// ---- DUTs/IO/Boxes/KL_C7B8B3CA.TcDUT
{attribute 'GeneratedUsingTerminal: KL3351-0003'}
{attribute addProperty BoxType "KL3351-0003"}
{attribute addProperty Description ""}
{attribute addProperty Physics ""}
{attribute addProperty Id "Channel_1AT %Q*Channel_0514A8FA0"}
{attribute addProperty CRC "3350770634"}
{attribute addProperty Size "0"}
TYPE KL_C7B8B3CA :
STRUCT
	{attribute addProperty Name "Channel_1"}
	Channel_1 : Channel_0514A8FA;
END_STRUCT
END_TYPE

// ---- DUTs/IO/Boxes/KL3356_E004D4E2.TcDUT
{attribute 'GeneratedUsingTerminal: KL3356'}
{attribute addProperty BoxType "KL3356"}
{attribute addProperty Description ""}
{attribute addProperty Physics ""}
{attribute addProperty Id "Channel_1AT %Q*Channel_4E9D1E2D0"}
{attribute addProperty CRC "3758413026"}
{attribute addProperty Size "0"}
TYPE KL3356_E004D4E2 :
STRUCT
	{attribute addProperty Name "Channel_1"}
	Channel_1 : Channel_4E9D1E2D;
END_STRUCT
END_TYPE

// ---- DUTs/IO/Boxes/KL_EE1D4506.TcDUT
{attribute 'GeneratedUsingTerminal: KL3361-0001'}
{attribute addProperty BoxType "KL3361-0001"}
{attribute addProperty Description ""}
{attribute addProperty Physics ""}
{attribute addProperty Id "Channel_1AT %Q*Channel_3C1A65000"}
{attribute addProperty CRC "3994895622"}
{attribute addProperty Size "0"}
TYPE KL_EE1D4506 :
STRUCT
	{attribute addProperty Name "Channel_1"}
	Channel_1 : Channel_3C1A6500;
END_STRUCT
END_TYPE

// ---- DUTs/IO/Boxes/KL3361_73CB82BA.TcDUT
{attribute 'GeneratedUsingTerminal: KL3361'}
{attribute addProperty BoxType "KL3361"}
{attribute addProperty Description ""}
{attribute addProperty Physics ""}
{attribute addProperty Id "Channel_1AT %Q*Channel_78571FB40"}
{attribute addProperty CRC "1942717114"}
{attribute addProperty Size "0"}
TYPE KL3361_73CB82BA :
STRUCT
	{attribute addProperty Name "Channel_1"}
	Channel_1 : Channel_78571FB4;
END_STRUCT
END_TYPE

// ---- DUTs/IO/Boxes/KL_73CB82BA.TcDUT
{attribute 'GeneratedUsingTerminal: KL3361-0003'}
{attribute addProperty BoxType "KL3361-0003"}
{attribute addProperty Description ""}
{attribute addProperty Physics ""}
{attribute addProperty Id "Channel_1AT %Q*Channel_78571FB40"}
{attribute addProperty CRC "1942717114"}
{attribute addProperty Size "0"}
TYPE KL_73CB82BA :
STRUCT
	{attribute addProperty Name "Channel_1"}
	Channel_1 : Channel_78571FB4;
END_STRUCT
END_TYPE

// ---- DUTs/IO/Boxes/KL3362_E98BF8F1.TcDUT
{attribute 'GeneratedUsingTerminal: KL3362'}
{attribute addProperty BoxType "KL3362"}
{attribute addProperty Description ""}
{attribute addProperty Physics ""}
{attribute addProperty Id "Channel_1AT %Q*Channel_3C1A65000Channel_2AT %Q*Channel_3C1A65000"}
{attribute addProperty CRC "3918264561"}
{attribute addProperty Size "0"}
TYPE KL3362_E98BF8F1 :
STRUCT
	{attribute addProperty Name "Channel_1"}
	Channel_1 : Channel_3C1A6500;
	{attribute addProperty Name "Channel_2"}
	Channel_2 : Channel_3C1A6500;
END_STRUCT
END_TYPE

// ---- DUTs/IO/Boxes/KL6211_60136EA1.TcDUT
{attribute 'GeneratedUsingTerminal: KL6211'}
{attribute addProperty BoxType "KL6211"}
{attribute addProperty Description ""}
{attribute addProperty Physics ""}
{attribute addProperty Id "Channel_1AT %Q*Channel_879058310"}
{attribute addProperty CRC "1611886241"}
{attribute addProperty Size "0"}
TYPE KL6211_60136EA1 :
STRUCT
	{attribute addProperty Name "Channel_1"}
	Channel_1 : Channel_87905831;
END_STRUCT
END_TYPE

// ---- DUTs/IO/Boxes/KL_9AE543B6.TcDUT
{attribute 'GeneratedUsingTerminal: KL6211-0020'}
{attribute addProperty BoxType "KL6211-0020"}
{attribute addProperty Description ""}
{attribute addProperty Physics ""}
{attribute addProperty Id "Channel_1AT %Q*Channel_099BCCDA0"}
{attribute addProperty CRC "2598716342"}
{attribute addProperty Size "0"}
TYPE KL_9AE543B6 :
STRUCT
	{attribute addProperty Name "Channel_1"}
	Channel_1 : Channel_099BCCDA;
END_STRUCT
END_TYPE

// ---- DUTs/IO/Boxes/KL_FC0201B8.TcDUT
{attribute 'GeneratedUsingTerminal: KL6211-0002'}
{attribute addProperty BoxType "KL6211-0002"}
{attribute addProperty Description ""}
{attribute addProperty Physics ""}
{attribute addProperty Id "Channel_1AT %Q*Channel_82ADD0760"}
{attribute addProperty CRC "4227989944"}
{attribute addProperty Size "0"}
TYPE KL_FC0201B8 :
STRUCT
	{attribute addProperty Name "Channel_1"}
	Channel_1 : Channel_82ADD076;
END_STRUCT
END_TYPE

// ---- DUTs/IO/Boxes/KL_498D8863.TcDUT
{attribute 'GeneratedUsingTerminal: KL6211-0022'}
{attribute addProperty BoxType "KL6211-0022"}
{attribute addProperty Description ""}
{attribute addProperty Physics ""}
{attribute addProperty Id "Channel_1AT %Q*Channel_332F026B0"}
{attribute addProperty CRC "1234012259"}
{attribute addProperty Size "0"}
TYPE KL_498D8863 :
STRUCT
	{attribute addProperty Name "Channel_1"}
	Channel_1 : Channel_332F026B;
END_STRUCT
END_TYPE

// ---- DUTs/IO/Boxes/KL_71341691.TcDUT
{attribute 'GeneratedUsingTerminal: KL6211-0004'}
{attribute addProperty BoxType "KL6211-0004"}
{attribute addProperty Description ""}
{attribute addProperty Physics ""}
{attribute addProperty Id "Channel_1AT %Q*Channel_A6A8AB450"}
{attribute addProperty CRC "1899239057"}
{attribute addProperty Size "0"}
TYPE KL_71341691 :
STRUCT
	{attribute addProperty Name "Channel_1"}
	Channel_1 : Channel_A6A8AB45;
END_STRUCT
END_TYPE

// ---- DUTs/IO/Boxes/KL_2B11657C.TcDUT
{attribute 'GeneratedUsingTerminal: KL6211-0024'}
{attribute addProperty BoxType "KL6211-0024"}
{attribute addProperty Description ""}
{attribute addProperty Physics ""}
{attribute addProperty Id "Channel_1AT %Q*Channel_A42BCA5C0"}
{attribute addProperty CRC "722560380"}
{attribute addProperty Size "0"}
TYPE KL_2B11657C :
STRUCT
	{attribute addProperty Name "Channel_1"}
	Channel_1 : Channel_A42BCA5C;
END_STRUCT
END_TYPE

// ---- DUTs/IO/Boxes/KL6224_C0F107BD.TcDUT
{attribute 'GeneratedUsingTerminal: KL6224'}
{attribute addProperty BoxType "KL6224"}
{attribute addProperty Description ""}
{attribute addProperty Physics ""}
{attribute addProperty Id "Channel_1AT %Q*Channel_08506BCE0"}
{attribute addProperty CRC "3237021629"}
{attribute addProperty Size "0"}
TYPE KL6224_C0F107BD :
STRUCT
	{attribute addProperty Name "Channel_1"}
	Channel_1 : Channel_08506BCE;
END_STRUCT
END_TYPE

// ---- DUTs/IO/Boxes/KL_FC1E3393.TcDUT
{attribute 'GeneratedUsingTerminal: KL6224-0001'}
{attribute addProperty BoxType "KL6224-0001"}
{attribute addProperty Description ""}
{attribute addProperty Physics ""}
{attribute addProperty Id "Channel_1AT %Q*Channel_085338040"}
{attribute addProperty CRC "4229837715"}
{attribute addProperty Size "0"}
TYPE KL_FC1E3393 :
STRUCT
	{attribute addProperty Name "Channel_1"}
	Channel_1 : Channel_08533804;
END_STRUCT
END_TYPE

// ---- DUTs/IO/Boxes/KL_C51B1CB0.TcDUT
{attribute 'GeneratedUsingTerminal: KL6224-0002'}
{attribute addProperty BoxType "KL6224-0002"}
{attribute addProperty Description ""}
{attribute addProperty Physics ""}
{attribute addProperty Id "Channel_1AT %Q*Channel_A04AC4BD0"}
{attribute addProperty CRC "3306888368"}
{attribute addProperty Size "0"}
TYPE KL_C51B1CB0 :
STRUCT
	{attribute addProperty Name "Channel_1"}
	Channel_1 : Channel_A04AC4BD;
END_STRUCT
END_TYPE

// ---- DUTs/IO/Boxes/KL_7EC2CD64.TcDUT
{attribute 'GeneratedUsingTerminal: KL6224-0003'}
{attribute addProperty BoxType "KL6224-0003"}
{attribute addProperty Description ""}
{attribute addProperty Physics ""}
{attribute addProperty Id "Channel_1AT %Q*Channel_779103830"}
{attribute addProperty CRC "2126695780"}
{attribute addProperty Size "0"}
TYPE KL_7EC2CD64 :
STRUCT
	{attribute addProperty Name "Channel_1"}
	Channel_1 : Channel_77910383;
END_STRUCT
END_TYPE

// ---- DUTs/IO/Boxes/KL_3829421A.TcDUT
{attribute 'GeneratedUsingTerminal: KL6301-0002'}
{attribute addProperty BoxType "KL6301-0002"}
{attribute addProperty Description ""}
{attribute addProperty Physics ""}
{attribute addProperty Id "Channel_1AT %Q*Channel_9BC0092E0"}
{attribute addProperty CRC "942227994"}
{attribute addProperty Size "0"}
TYPE KL_3829421A :
STRUCT
	{attribute addProperty Name "Channel_1"}
	Channel_1 : Channel_9BC0092E;
END_STRUCT
END_TYPE

// ---- DUTs/IO/Boxes/KL_9116C2C1.TcDUT
{attribute 'GeneratedUsingTerminal: KL6401-0002'}
{attribute addProperty BoxType "KL6401-0002"}
{attribute addProperty Description ""}
{attribute addProperty Physics ""}
{attribute addProperty Id "Channel_1AT %Q*Channel_7606D9890"}
{attribute addProperty CRC "2434187969"}
{attribute addProperty Size "0"}
TYPE KL_9116C2C1 :
STRUCT
	{attribute addProperty Name "Channel_1"}
	Channel_1 : Channel_7606D989;
END_STRUCT
END_TYPE

// ---- DUTs/IO/Boxes/KL6551_528AE398.TcDUT
{attribute 'GeneratedUsingTerminal: KL6551'}
{attribute addProperty BoxType "KL6551"}
{attribute addProperty Description ""}
{attribute addProperty Physics ""}
{attribute addProperty Id "Channel_1AT %Q*Channel_6931CC5B0"}
{attribute addProperty CRC "1384833944"}
{attribute addProperty Size "0"}
TYPE KL6551_528AE398 :
STRUCT
	{attribute addProperty Name "Channel_1"}
	Channel_1 : Channel_6931CC5B;
END_STRUCT
END_TYPE

// ---- DUTs/IO/Boxes/KL_3325E583.TcDUT
{attribute 'GeneratedUsingTerminal: KL6581-0002'}
{attribute addProperty BoxType "KL6581-0002"}
{attribute addProperty Description ""}
{attribute addProperty Physics ""}
{attribute addProperty Id "Channel_1AT %Q*Channel_F7FDEFA00"}
{attribute addProperty CRC "858121603"}
{attribute addProperty Size "0"}
TYPE KL_3325E583 :
STRUCT
	{attribute addProperty Name "Channel_1"}
	Channel_1 : Channel_F7FDEFA0;
END_STRUCT
END_TYPE

// ---- DUTs/IO/Boxes/KL_528AE398.TcDUT
{attribute 'GeneratedUsingTerminal: KL6771-0002'}
{attribute addProperty BoxType "KL6771-0002"}
{attribute addProperty Description ""}
{attribute addProperty Physics ""}
{attribute addProperty Id "Channel_1AT %Q*Channel_6931CC5B0"}
{attribute addProperty CRC "1384833944"}
{attribute addProperty Size "0"}
TYPE KL_528AE398 :
STRUCT
	{attribute addProperty Name "Channel_1"}
	Channel_1 : Channel_6931CC5B;
END_STRUCT
END_TYPE

// ---- DUTs/IO/Boxes/KL6781_BE595CA2.TcDUT
{attribute 'GeneratedUsingTerminal: KL6781'}
{attribute addProperty BoxType "KL6781"}
{attribute addProperty Description ""}
{attribute addProperty Physics ""}
{attribute addProperty Id "Channel_1AT %Q*Channel_A1C14FB40"}
{attribute addProperty CRC "3193527458"}
{attribute addProperty Size "0"}
TYPE KL6781_BE595CA2 :
STRUCT
	{attribute addProperty Name "Channel_1"}
	Channel_1 : Channel_A1C14FB4;
END_STRUCT
END_TYPE

// ---- DUTs/IO/Boxes/KL6811_6148C904.TcDUT
{attribute 'GeneratedUsingTerminal: KL6811'}
{attribute addProperty BoxType "KL6811"}
{attribute addProperty Description ""}
{attribute addProperty Physics ""}
{attribute addProperty Id "Channel_1AT %Q*Channel_6576A6810"}
{attribute addProperty CRC "1632160004"}
{attribute addProperty Size "0"}
TYPE KL6811_6148C904 :
STRUCT
	{attribute addProperty Name "Channel_1"}
	Channel_1 : Channel_6576A681;
END_STRUCT
END_TYPE

// ---- DUTs/IO/Boxes/KL6821_F77C82D2.TcDUT
{attribute 'GeneratedUsingTerminal: KL6821'}
{attribute addProperty BoxType "KL6821"}
{attribute addProperty Description ""}
{attribute addProperty Physics ""}
{attribute addProperty Id "Channel_1AT %Q*Channel_A4B48F2D0"}
{attribute addProperty CRC "4152132306"}
{attribute addProperty Size "0"}
TYPE KL6821_F77C82D2 :
STRUCT
	{attribute addProperty Name "Channel_1"}
	Channel_1 : Channel_A4B48F2D;
END_STRUCT
END_TYPE

// ---- DUTs/IO/Boxes/KL6831_BE595CA2.TcDUT
{attribute 'GeneratedUsingTerminal: KL6831'}
{attribute addProperty BoxType "KL6831"}
{attribute addProperty Description ""}
{attribute addProperty Physics ""}
{attribute addProperty Id "Channel_1AT %Q*Channel_A1C14FB40"}
{attribute addProperty CRC "3193527458"}
{attribute addProperty Size "0"}
TYPE KL6831_BE595CA2 :
STRUCT
	{attribute addProperty Name "Channel_1"}
	Channel_1 : Channel_A1C14FB4;
END_STRUCT
END_TYPE

// ---- DUTs/IO/Boxes/KL6841_BE595CA2.TcDUT
{attribute 'GeneratedUsingTerminal: KL6841'}
{attribute addProperty BoxType "KL6841"}
{attribute addProperty Description ""}
{attribute addProperty Physics ""}
{attribute addProperty Id "Channel_1AT %Q*Channel_A1C14FB40"}
{attribute addProperty CRC "3193527458"}
{attribute addProperty Size "0"}
TYPE KL6841_BE595CA2 :
STRUCT
	{attribute addProperty Name "Channel_1"}
	Channel_1 : Channel_A1C14FB4;
END_STRUCT
END_TYPE

// ---- DUTs/IO/Boxes/KL6904_B938D612.TcDUT
{attribute 'GeneratedUsingTerminal: KL6904'}
{attribute addProperty BoxType "KL6904"}
{attribute addProperty Description ""}
{attribute addProperty Physics ""}
{attribute addProperty Id "Channel_1AT %Q*Channel_9E2936860"}
{attribute addProperty CRC "3107509778"}
{attribute addProperty Size "0"}
TYPE KL6904_B938D612 :
STRUCT
	{attribute addProperty Name "Channel_1"}
	Channel_1 : Channel_9E293686;
END_STRUCT
END_TYPE

// ---- DUTs/IO/Boxes/KL_921B772D.TcDUT
{attribute 'GeneratedUsingTerminal: KL6904-0001'}
{attribute addProperty BoxType "KL6904-0001"}
{attribute addProperty Description ""}
{attribute addProperty Physics ""}
{attribute addProperty Id "Channel_1AT %Q*Channel_F84AC14F0"}
{attribute addProperty CRC "2451273517"}
{attribute addProperty Size "0"}
TYPE KL_921B772D :
STRUCT
	{attribute addProperty Name "Channel_1"}
	Channel_1 : Channel_F84AC14F;
END_STRUCT
END_TYPE

// ---- DUTs/IO/Boxes/KL_779990DF.TcDUT
{attribute 'GeneratedUsingTerminal: KL8001-0002'}
{attribute addProperty BoxType "KL8001-0002"}
{attribute addProperty Description ""}
{attribute addProperty Physics ""}
{attribute addProperty Id "Channel_1AT %Q*Channel_2F3145090"}
{attribute addProperty CRC "2006552799"}
{attribute addProperty Size "0"}
TYPE KL_779990DF :
STRUCT
	{attribute addProperty Name "Channel_1"}
	Channel_1 : Channel_2F314509;
END_STRUCT
END_TYPE

// ---- DUTs/IO/Boxes/KL8001_7761653A.TcDUT
{attribute 'GeneratedUsingTerminal: KL8001'}
{attribute addProperty BoxType "KL8001"}
{attribute addProperty Description ""}
{attribute addProperty Physics ""}
{attribute addProperty Id "Channel_1AT %Q*Channel_D9D488070"}
{attribute addProperty CRC "2002871610"}
{attribute addProperty Size "0"}
TYPE KL8001_7761653A :
STRUCT
	{attribute addProperty Name "Channel_1"}
	Channel_1 : Channel_D9D48807;
END_STRUCT
END_TYPE

// ---- DUTs/IO/Boxes/KL8519_8C34650F.TcDUT
{attribute 'GeneratedUsingTerminal: KL8519'}
{attribute addProperty BoxType "KL8519"}
{attribute addProperty Description ""}
{attribute addProperty Physics ""}
{attribute addProperty Id "Channel_1AT %Q*Channel_D13646E30"}
{attribute addProperty CRC "2352243983"}
{attribute addProperty Size "0"}
TYPE KL8519_8C34650F :
STRUCT
	{attribute addProperty Name "Channel_1"}
	Channel_1 : Channel_D13646E3;
END_STRUCT
END_TYPE

// ---- DUTs/IO/Boxes/KL8524_A4B9216E.TcDUT
{attribute 'GeneratedUsingTerminal: KL8524'}
{attribute addProperty BoxType "KL8524"}
{attribute addProperty Description ""}
{attribute addProperty Physics ""}
{attribute addProperty Id "Channel_1AT %Q*Channel_3263D8D50"}
{attribute addProperty CRC "2763596142"}
{attribute addProperty Size "0"}
TYPE KL8524_A4B9216E :
STRUCT
	{attribute addProperty Name "Channel_1"}
	Channel_1 : Channel_3263D8D5;
END_STRUCT
END_TYPE

// ---- DUTs/IO/Boxes/KL8528_73A97EC1.TcDUT
{attribute 'GeneratedUsingTerminal: KL8528'}
{attribute addProperty BoxType "KL8528"}
{attribute addProperty Description ""}
{attribute addProperty Physics ""}
{attribute addProperty Id "Channel_1AT %Q*Channel_D490E9730"}
{attribute addProperty CRC "1940487873"}
{attribute addProperty Size "0"}
TYPE KL8528_73A97EC1 :
STRUCT
	{attribute addProperty Name "Channel_1"}
	Channel_1 : Channel_D490E973;
END_STRUCT
END_TYPE

// ---- DUTs/IO/Boxes/KL8548_23451728.TcDUT
{attribute 'GeneratedUsingTerminal: KL8548'}
{attribute addProperty BoxType "KL8548"}
{attribute addProperty Description ""}
{attribute addProperty Physics ""}
{attribute addProperty Id "Channel_1AT %Q*Channel_6576A6810Channel_2AT %Q*Channel_6576A6810Channel_3AT %Q*Channel_6576A6810Channel_4AT %Q*Channel_6576A6810Channel_5AT %Q*Channel_6576A6810Channel_6AT %Q*Channel_6576A6810Channel_7AT %Q*Channel_6576A6810Channel_8AT %Q*Channel_6576A6810"}
{attribute addProperty CRC "591730472"}
{attribute addProperty Size "0"}
TYPE KL8548_23451728 :
STRUCT
	{attribute addProperty Name "Channel_1"}
	Channel_1 : Channel_6576A681;
	{attribute addProperty Name "Channel_2"}
	Channel_2 : Channel_6576A681;
	{attribute addProperty Name "Channel_3"}
	Channel_3 : Channel_6576A681;
	{attribute addProperty Name "Channel_4"}
	Channel_4 : Channel_6576A681;
	{attribute addProperty Name "Channel_5"}
	Channel_5 : Channel_6576A681;
	{attribute addProperty Name "Channel_6"}
	Channel_6 : Channel_6576A681;
	{attribute addProperty Name "Channel_7"}
	Channel_7 : Channel_6576A681;
	{attribute addProperty Name "Channel_8"}
	Channel_8 : Channel_6576A681;
END_STRUCT
END_TYPE

// ---- DUTs/IO/Boxes/KL8610_C571D068.TcDUT
{attribute 'GeneratedUsingTerminal: KL8610'}
{attribute addProperty BoxType "KL8610"}
{attribute addProperty Description ""}
{attribute addProperty Physics ""}
{attribute addProperty Id "KL8601_1AT %Q*KL_6576A6810"}
{attribute addProperty CRC "3312570472"}
{attribute addProperty Size "0"}
TYPE KL8610_C571D068 :
STRUCT
	{attribute addProperty Name "KL8601_1"}
	KL8601_1 : KL_6576A681;
END_STRUCT
END_TYPE

// ---- DUTs/IO/Boxes/KL_5A83E84C.TcDUT
{attribute 'GeneratedUsingTerminal: KL8610-0001'}
{attribute addProperty BoxType "KL8610-0001"}
{attribute addProperty Description ""}
{attribute addProperty Physics ""}
{attribute addProperty Id "KL8601_1AT %Q*KL_6576A6810KL8601_2AT %Q*KL_6576A6810"}
{attribute addProperty CRC "1518594124"}
{attribute addProperty Size "0"}
TYPE KL_5A83E84C :
STRUCT
	{attribute addProperty Name "KL8601_1"}
	KL8601_1 : KL_6576A681;
	{attribute addProperty Name "KL8601_2"}
	KL8601_2 : KL_6576A681;
END_STRUCT
END_TYPE

// ---- DUTs/IO/Boxes/KL_BF4AA06C.TcDUT
{attribute 'GeneratedUsingTerminal: KL8610-0002'}
{attribute addProperty BoxType "KL8610-0002"}
{attribute addProperty Description ""}
{attribute addProperty Physics ""}
{attribute addProperty Id "KL8601_1AT %Q*KL_6576A6810KL8601_2AT %Q*KL_6576A6810KL8601_3AT %Q*KL_6576A6810"}
{attribute addProperty CRC "3209338988"}
{attribute addProperty Size "0"}
TYPE KL_BF4AA06C :
STRUCT
	{attribute addProperty Name "KL8601_1"}
	KL8601_1 : KL_6576A681;
	{attribute addProperty Name "KL8601_2"}
	KL8601_2 : KL_6576A681;
	{attribute addProperty Name "KL8601_3"}
	KL8601_3 : KL_6576A681;
END_STRUCT
END_TYPE

// ---- DUTs/IO/Boxes/KL_7485E925.TcDUT
{attribute 'GeneratedUsingTerminal: KL8610-0003'}
{attribute addProperty BoxType "KL8610-0003"}
{attribute addProperty Description ""}
{attribute addProperty Physics ""}
{attribute addProperty Id "KL8601_1AT %Q*KL_6576A6810KL8601_2AT %Q*KL_6576A6810KL8601_3AT %Q*KL_6576A6810KL8601_4AT %Q*KL_6576A6810"}
{attribute addProperty CRC "1954933029"}
{attribute addProperty Size "0"}
TYPE KL_7485E925 :
STRUCT
	{attribute addProperty Name "KL8601_1"}
	KL8601_1 : KL_6576A681;
	{attribute addProperty Name "KL8601_2"}
	KL8601_2 : KL_6576A681;
	{attribute addProperty Name "KL8601_3"}
	KL8601_3 : KL_6576A681;
	{attribute addProperty Name "KL8601_4"}
	KL8601_4 : KL_6576A681;
END_STRUCT
END_TYPE

// ---- DUTs/IO/Boxes/KL_372C6BEC.TcDUT
{attribute 'GeneratedUsingTerminal: KL8610-0004'}
{attribute addProperty BoxType "KL8610-0004"}
{attribute addProperty Description ""}
{attribute addProperty Physics ""}
{attribute addProperty Id "KL8601_1AT %Q*KL_6576A6810KL8601_2AT %Q*KL_6576A6810KL8601_3AT %Q*KL_6576A6810KL8601_4AT %Q*KL_6576A6810KL8601_5AT %Q*KL_6576A6810"}
{attribute addProperty CRC "925658092"}
{attribute addProperty Size "0"}
TYPE KL_372C6BEC :
STRUCT
	{attribute addProperty Name "KL8601_1"}
	KL8601_1 : KL_6576A681;
	{attribute addProperty Name "KL8601_2"}
	KL8601_2 : KL_6576A681;
	{attribute addProperty Name "KL8601_3"}
	KL8601_3 : KL_6576A681;
	{attribute addProperty Name "KL8601_4"}
	KL8601_4 : KL_6576A681;
	{attribute addProperty Name "KL8601_5"}
	KL8601_5 : KL_6576A681;
END_STRUCT
END_TYPE

// ---- DUTs/IO/Boxes/KL_2E5CD6C8.TcDUT
{attribute 'GeneratedUsingTerminal: KL8610-0005'}
{attribute addProperty BoxType "KL8610-0005"}
{attribute addProperty Description ""}
{attribute addProperty Physics ""}
{attribute addProperty Id "KL8601_1AT %Q*KL_6576A6810KL8601_2AT %Q*KL_6576A6810KL8601_3AT %Q*KL_6576A6810KL8601_4AT %Q*KL_6576A6810KL8601_5AT %Q*KL_6576A6810KL8601_6AT %Q*KL_6576A6810"}
{attribute addProperty CRC "777836232"}
{attribute addProperty Size "0"}
TYPE KL_2E5CD6C8 :
STRUCT
	{attribute addProperty Name "KL8601_1"}
	KL8601_1 : KL_6576A681;
	{attribute addProperty Name "KL8601_2"}
	KL8601_2 : KL_6576A681;
	{attribute addProperty Name "KL8601_3"}
	KL8601_3 : KL_6576A681;
	{attribute addProperty Name "KL8601_4"}
	KL8601_4 : KL_6576A681;
	{attribute addProperty Name "KL8601_5"}
	KL8601_5 : KL_6576A681;
	{attribute addProperty Name "KL8601_6"}
	KL8601_6 : KL_6576A681;
END_STRUCT
END_TYPE

// ---- DUTs/IO/Boxes/KL_68BDE1E9.TcDUT
{attribute 'GeneratedUsingTerminal: KL8610-0006'}
{attribute addProperty BoxType "KL8610-0006"}
{attribute addProperty Description ""}
{attribute addProperty Physics ""}
{attribute addProperty Id "KL8601_1AT %Q*KL_6576A6810KL8601_2AT %Q*KL_6576A6810KL8601_3AT %Q*KL_6576A6810KL8601_4AT %Q*KL_6576A6810KL8601_5AT %Q*KL_6576A6810KL8601_6AT %Q*KL_6576A6810KL8601_7AT %Q*KL_6576A6810"}
{attribute addProperty CRC "1757274601"}
{attribute addProperty Size "0"}
TYPE KL_68BDE1E9 :
STRUCT
	{attribute addProperty Name "KL8601_1"}
	KL8601_1 : KL_6576A681;
	{attribute addProperty Name "KL8601_2"}
	KL8601_2 : KL_6576A681;
	{attribute addProperty Name "KL8601_3"}
	KL8601_3 : KL_6576A681;
	{attribute addProperty Name "KL8601_4"}
	KL8601_4 : KL_6576A681;
	{attribute addProperty Name "KL8601_5"}
	KL8601_5 : KL_6576A681;
	{attribute addProperty Name "KL8601_6"}
	KL8601_6 : KL_6576A681;
	{attribute addProperty Name "KL8601_7"}
	KL8601_7 : KL_6576A681;
END_STRUCT
END_TYPE

// ---- DUTs/IO/Boxes/KL_84AAE8B6.TcDUT
{attribute 'GeneratedUsingTerminal: KL8610-0007'}
{attribute addProperty BoxType "KL8610-0007"}
{attribute addProperty Description ""}
{attribute addProperty Physics ""}
{attribute addProperty Id "KL8601_1AT %Q*KL_6576A6810KL8601_2AT %Q*KL_6576A6810KL8601_3AT %Q*KL_6576A6810KL8601_4AT %Q*KL_6576A6810KL8601_5AT %Q*KL_6576A6810KL8601_6AT %Q*KL_6576A6810KL8601_7AT %Q*KL_6576A6810KL8601_8AT %Q*KL_6576A6810"}
{attribute addProperty CRC "2225793206"}
{attribute addProperty Size "0"}
TYPE KL_84AAE8B6 :
STRUCT
	{attribute addProperty Name "KL8601_1"}
	KL8601_1 : KL_6576A681;
	{attribute addProperty Name "KL8601_2"}
	KL8601_2 : KL_6576A681;
	{attribute addProperty Name "KL8601_3"}
	KL8601_3 : KL_6576A681;
	{attribute addProperty Name "KL8601_4"}
	KL8601_4 : KL_6576A681;
	{attribute addProperty Name "KL8601_5"}
	KL8601_5 : KL_6576A681;
	{attribute addProperty Name "KL8601_6"}
	KL8601_6 : KL_6576A681;
	{attribute addProperty Name "KL8601_7"}
	KL8601_7 : KL_6576A681;
	{attribute addProperty Name "KL8601_8"}
	KL8601_8 : KL_6576A681;
END_STRUCT
END_TYPE

// ---- DUTs/IO/Boxes/KL9110_8BEE55F2.TcDUT
{attribute 'GeneratedUsingTerminal: KL9110'}
{attribute addProperty BoxType "KL9110"}
{attribute addProperty Description ""}
{attribute addProperty Physics ""}
{attribute addProperty Id "Channel_1AT %I*Channel_64AAC8C70"}
{attribute addProperty CRC "2347652594"}
{attribute addProperty Size "0"}
TYPE KL9110_8BEE55F2 :
STRUCT
	{attribute addProperty Name "Channel_1"}
	Channel_1 : Channel_64AAC8C7;
END_STRUCT
END_TYPE

// ---- DUTs/IO/Boxes/KL9160_8BEE55F2.TcDUT
{attribute 'GeneratedUsingTerminal: KL9160'}
{attribute addProperty BoxType "KL9160"}
{attribute addProperty Description ""}
{attribute addProperty Physics ""}
{attribute addProperty Id "Channel_1AT %I*Channel_64AAC8C70"}
{attribute addProperty CRC "2347652594"}
{attribute addProperty Size "0"}
TYPE KL9160_8BEE55F2 :
STRUCT
	{attribute addProperty Name "Channel_1"}
	Channel_1 : Channel_64AAC8C7;
END_STRUCT
END_TYPE

// ---- DUTs/IO/Boxes/KL9191_962A24DF.TcDUT
{attribute 'GeneratedUsingTerminal: KL9191'}
{attribute addProperty BoxType "KL9191"}
{attribute addProperty Description ""}
{attribute addProperty Physics ""}
{attribute addProperty Id "Channel_1AT %Q*Channel_471FAA5C0"}
{attribute addProperty CRC "2519344351"}
{attribute addProperty Size "0"}
TYPE KL9191_962A24DF :
STRUCT
	{attribute addProperty Name "Channel_1"}
	Channel_1 : Channel_471FAA5C;
END_STRUCT
END_TYPE

// ---- DUTs/IO/Boxes/KL9210_8BEE55F2.TcDUT
{attribute 'GeneratedUsingTerminal: KL9210'}
{attribute addProperty BoxType "KL9210"}
{attribute addProperty Description ""}
{attribute addProperty Physics ""}
{attribute addProperty Id "Channel_1AT %I*Channel_64AAC8C70"}
{attribute addProperty CRC "2347652594"}
{attribute addProperty Size "0"}
TYPE KL9210_8BEE55F2 :
STRUCT
	{attribute addProperty Name "Channel_1"}
	Channel_1 : Channel_64AAC8C7;
END_STRUCT
END_TYPE

// ---- DUTs/IO/Boxes/KL9260_8BEE55F2.TcDUT
{attribute 'GeneratedUsingTerminal: KL9260'}
{attribute addProperty BoxType "KL9260"}
{attribute addProperty Description ""}
{attribute addProperty Physics ""}
{attribute addProperty Id "Channel_1AT %I*Channel_64AAC8C70"}
{attribute addProperty CRC "2347652594"}
{attribute addProperty Size "0"}
TYPE KL9260_8BEE55F2 :
STRUCT
	{attribute addProperty Name "Channel_1"}
	Channel_1 : Channel_64AAC8C7;
END_STRUCT
END_TYPE

// ---- DUTs/IO/Boxes/KL_E4BD2B38.TcDUT
{attribute 'GeneratedUsingTerminal: KL9505-0010'}
{attribute addProperty BoxType "KL9505-0010"}
{attribute addProperty Description ""}
{attribute addProperty Physics ""}
{attribute addProperty Id "Diag_1AT %I*Diag_1F4F45730"}
{attribute addProperty CRC "3837602616"}
{attribute addProperty Size "0"}
TYPE KL_E4BD2B38 :
STRUCT
	{attribute addProperty Name "Diag_1"}
	Diag_1 : Diag_1F4F4573;
END_STRUCT
END_TYPE

// ---- DUTs/IO/Boxes/KL9528_8C984603.TcDUT
{attribute 'GeneratedUsingTerminal: KL9528'}
{attribute addProperty BoxType "KL9528"}
{attribute addProperty Description ""}
{attribute addProperty Physics ""}
{attribute addProperty Id "Channel_1AT %Q*Channel_0029832E0"}
{attribute addProperty CRC "2358789635"}
{attribute addProperty Size "0"}
TYPE KL9528_8C984603 :
STRUCT
	{attribute addProperty Name "Channel_1"}
	Channel_1 : Channel_0029832E;
END_STRUCT
END_TYPE

// ---- DUTs/IO/Boxes/KL9999_7A10A7F6.TcDUT
{attribute 'GeneratedUsingTerminal: KL9999'}
{attribute addProperty BoxType "KL9999"}
{attribute addProperty Description ""}
{attribute addProperty Physics ""}
{attribute addProperty Id "Channel_1AT %Q*Channel_126527430"}
{attribute addProperty CRC "2047911926"}
{attribute addProperty Size "0"}
TYPE KL9999_7A10A7F6 :
STRUCT
	{attribute addProperty Name "Channel_1"}
	Channel_1 : Channel_12652743;
END_STRUCT
END_TYPE

// ---- DUTs/IO/Devices/SyncUnitTask_2D604ED5.TcDUT
{attribute 'GeneratedUsingTerminal: IODEVICETYPE_ETHERCATPROT'}
{attribute addProperty BoxType "IODEVICETYPE_ETHERCATPROT"}
{attribute addProperty Id "WcStateAT %I*WcState_0B2B16F91InfoDataAT %I*InfoData_2A97D6CF8"}
{attribute addProperty CRC "761286357"}
{attribute addProperty Size "9"}
TYPE SyncUnitTask_2D604ED5 :
STRUCT
	{attribute addProperty Name "WcState"}
	WcState : WcState_0B2B16F9;
	{attribute addProperty Name "InfoData"}
	InfoData : InfoData_2A97D6CF;
END_STRUCT
END_TYPE

// ---- DUTs/IO/Devices/SyncUnitTasks_6FEB8257.TcDUT
{attribute 'GeneratedUsingTerminal: '}
{attribute addProperty BoxType ""}
{attribute addProperty Id "unreferencedAT %I*SyncUnitTask_2D604ED59PlcTaskAT %I*SyncUnitTask_2D604ED59"}
{attribute addProperty CRC "1877705303"}
{attribute addProperty Size "18"}
TYPE SyncUnitTasks_6FEB8257 :
STRUCT
	{attribute addProperty Name "unreferenced"}
	unreferenced : SyncUnitTask_2D604ED5;
	{attribute addProperty Name "PlcTask"}
	PlcTask : SyncUnitTask_2D604ED5;
END_STRUCT
END_TYPE

// ---- DUTs/IO/Devices/SyncUnits_99E584AF.TcDUT
{attribute 'GeneratedUsingTerminal: '}
{attribute addProperty BoxType ""}
{attribute addProperty Id "_defaultAT %I*SyncUnitTasks_6FEB825718"}
{attribute addProperty CRC "2581955759"}
{attribute addProperty Size "18"}
TYPE SyncUnits_99E584AF :
STRUCT
	{attribute addProperty Name "_default"}
	_default : SyncUnitTasks_6FEB8257;
END_STRUCT
END_TYPE

// ---- DUTs/IO/Topology/A_0014_BK1250_0000_0000_09E1EB45.TcDUT
{attribute 'GeneratedUsingTerminal: BK1250-0000-0000'}
{attribute addProperty BoxType "BK1250-0000-0000"}
{attribute addProperty Id "Term_397_KL1002KL1002_BB38DA8F0"}
{attribute addProperty CRC "165800773"}
{attribute addProperty Size "0"}
{attribute addProperty Name "A_0014(BK1250-0000-0000)"}
TYPE A_0014_BK1250_0000_0000_09E1EB45 EXTENDS BK1250_A2FCADE7 :
STRUCT
	{attribute addProperty Name "Term_397_KL1002"}
	Term_397_KL1002 : KL1002_BB38DA8F;
END_STRUCT
END_TYPE

// ---- DUTs/IO/Topology/Beckhoff_BKxxxxsub_EK1100_59A46924.TcDUT
{attribute 'GeneratedUsingTerminal: EK1100-0000-0018'}
{attribute addProperty BoxType "EK1100-0000-0018"}
{attribute addProperty Id "A_0014_BK1250_0000_0000A_0014_BK1250_0000_0000_09E1EB450"}
{attribute addProperty CRC "1503947044"}
{attribute addProperty Size "0"}
{attribute addProperty Name "Beckhoff BKxxxxsub EK1100"}
TYPE Beckhoff_BKxxxxsub_EK1100_59A46924 EXTENDS EK1100_1FC0878B :
STRUCT
	{attribute addProperty Name "A_0014(BK1250-0000-0000)"}
	{attribute addProperty PreviousPort "Beckhoff BKxxxxsub EK1100 : B"}
	A_0014_BK1250_0000_0000 : A_0014_BK1250_0000_0000_09E1EB45;
END_STRUCT
END_TYPE

// ---- DUTs/IO/Topology/A_0001_BK1120_0000_0000_205E6559.TcDUT
{attribute 'GeneratedUsingTerminal: BK1120-0000-0000'}
{attribute addProperty BoxType "BK1120-0000-0000"}
{attribute addProperty Id "Term_374_KL1002KL1002_BB38DA8F0"}
{attribute addProperty CRC "543057241"}
{attribute addProperty Size "0"}
{attribute addProperty Name "A_0001(BK1120-0000-0000)"}
TYPE A_0001_BK1120_0000_0000_205E6559 EXTENDS BK1120_6D44499E :
STRUCT
	{attribute addProperty Name "Term_374_KL1002"}
	Term_374_KL1002 : KL1002_BB38DA8F;
END_STRUCT
END_TYPE

// ---- DUTs/IO/Topology/A_0002_BK1120_0000_0001_76F1F8EB.TcDUT
{attribute 'GeneratedUsingTerminal: BK1120-0000-0001'}
{attribute addProperty BoxType "BK1120-0000-0001"}
{attribute addProperty Id "Term_375_KL1002KL1002_BB38DA8F0"}
{attribute addProperty CRC "1995569387"}
{attribute addProperty Size "0"}
{attribute addProperty Name "A_0002(BK1120-0000-0001)"}
TYPE A_0002_BK1120_0000_0001_76F1F8EB EXTENDS BK1120_A2FCADE7 :
STRUCT
	{attribute addProperty Name "Term_375_KL1002"}
	Term_375_KL1002 : KL1002_BB38DA8F;
END_STRUCT
END_TYPE

// ---- DUTs/IO/Topology/A_0003_BK1120_0000_0016_8D015E3D.TcDUT
{attribute 'GeneratedUsingTerminal: BK1120-0000-0016'}
{attribute addProperty BoxType "BK1120-0000-0016"}
{attribute addProperty Id "Term_376_KL1002KL1002_BB38DA8F0"}
{attribute addProperty CRC "2365677117"}
{attribute addProperty Size "0"}
{attribute addProperty Name "A_0003(BK1120-0000-0016)"}
TYPE A_0003_BK1120_0000_0016_8D015E3D EXTENDS BK1120_A2FCADE7 :
STRUCT
	{attribute addProperty Name "Term_376_KL1002"}
	Term_376_KL1002 : KL1002_BB38DA8F;
END_STRUCT
END_TYPE

// ---- DUTs/IO/Topology/A_0004_BK1120_0000_0017_DBAEC38F.TcDUT
{attribute 'GeneratedUsingTerminal: BK1120-0000-0017'}
{attribute addProperty BoxType "BK1120-0000-0017"}
{attribute addProperty Id "Term_377_KL1002KL1002_BB38DA8F0"}
{attribute addProperty CRC "3685663631"}
{attribute addProperty Size "0"}
{attribute addProperty Name "A_0004(BK1120-0000-0017)"}
TYPE A_0004_BK1120_0000_0017_DBAEC38F EXTENDS BK1120_A2FCADE7 :
STRUCT
	{attribute addProperty Name "Term_377_KL1002"}
	Term_377_KL1002 : KL1002_BB38DA8F;
END_STRUCT
END_TYPE

// ---- DUTs/IO/Topology/A_0005_BK1120_0000_0018_C2DFD8D8.TcDUT
{attribute 'GeneratedUsingTerminal: BK1120-0000-0018'}
{attribute addProperty BoxType "BK1120-0000-0018"}
{attribute addProperty Id "Term_378_KL1002KL1002_BB38DA8F0"}
{attribute addProperty CRC "3269449944"}
{attribute addProperty Size "0"}
{attribute addProperty Name "A_0005(BK1120-0000-0018)"}
TYPE A_0005_BK1120_0000_0018_C2DFD8D8 EXTENDS BK1120_A2FCADE7 :
STRUCT
	{attribute addProperty Name "Term_378_KL1002"}
	Term_378_KL1002 : KL1002_BB38DA8F;
END_STRUCT
END_TYPE

// ---- DUTs/IO/Topology/A_0006_BK1120_0000_0019_9470456A.TcDUT
{attribute 'GeneratedUsingTerminal: BK1120-0000-0019'}
{attribute addProperty BoxType "BK1120-0000-0019"}
{attribute addProperty Id "Term_379_KL1002KL1002_BB38DA8F0"}
{attribute addProperty CRC "2490385770"}
{attribute addProperty Size "0"}
{attribute addProperty Name "A_0006(BK1120-0000-0019)"}
TYPE A_0006_BK1120_0000_0019_9470456A EXTENDS BK1120_A2FCADE7 :
STRUCT
	{attribute addProperty Name "Term_379_KL1002"}
	Term_379_KL1002 : KL1002_BB38DA8F;
END_STRUCT
END_TYPE

// ---- DUTs/IO/Topology/A_0007_BK1120_0000_0020_61E27259.TcDUT
{attribute 'GeneratedUsingTerminal: BK1120-0000-0020'}
{attribute addProperty BoxType "BK1120-0000-0020"}
{attribute addProperty Id "Term_380_KL1002KL1002_BB38DA8F0"}
{attribute addProperty CRC "1642230361"}
{attribute addProperty Size "0"}
{attribute addProperty Name "A_0007(BK1120-0000-0020)"}
TYPE A_0007_BK1120_0000_0020_61E27259 EXTENDS BK1120_A2FCADE7 :
STRUCT
	{attribute addProperty Name "Term_380_KL1002"}
	Term_380_KL1002 : KL1002_BB38DA8F;
END_STRUCT
END_TYPE

// ---- DUTs/IO/Topology/A_0008_BK1120_0000_0021_374DEFEB.TcDUT
{attribute 'GeneratedUsingTerminal: BK1120-0000-0021'}
{attribute addProperty BoxType "BK1120-0000-0021"}
{attribute addProperty Id "Term_381_KL1002KL1002_BB38DA8F0"}
{attribute addProperty CRC "927854571"}
{attribute addProperty Size "0"}
{attribute addProperty Name "A_0008(BK1120-0000-0021)"}
TYPE A_0008_BK1120_0000_0021_374DEFEB EXTENDS BK1120_A2FCADE7 :
STRUCT
	{attribute addProperty Name "Term_381_KL1002"}
	Term_381_KL1002 : KL1002_BB38DA8F;
END_STRUCT
END_TYPE

// ---- DUTs/IO/Topology/A_0009_CPXXXX_BK1150_0016_CCBD493D.TcDUT
{attribute 'GeneratedUsingTerminal: CPXXXX-BK7902-0016'}
{attribute addProperty BoxType "CPXXXX-BK7902-0016"}
{attribute addProperty Id "Term_382_KL1002KL1002_BB38DA8F0"}
{attribute addProperty CRC "3434957117"}
{attribute addProperty Size "0"}
{attribute addProperty Name "A_0009(CPXXXX-BK1150-0016)"}
TYPE A_0009_CPXXXX_BK1150_0016_CCBD493D EXTENDS CPXXXX_A2FCADE7 :
STRUCT
	{attribute addProperty Name "Term_382_KL1002"}
	Term_382_KL1002 : KL1002_BB38DA8F;
END_STRUCT
END_TYPE

// ---- DUTs/IO/Topology/A_0010_BK1150_0000_0016_9A12D48F.TcDUT
{attribute 'GeneratedUsingTerminal: BK1150-0000-0016'}
{attribute addProperty BoxType "BK1150-0000-0016"}
{attribute addProperty Id "Term_383_KL1002KL1002_BB38DA8F0"}
{attribute addProperty CRC "2584925327"}
{attribute addProperty Size "0"}
{attribute addProperty Name "A_0010(BK1150-0000-0016)"}
TYPE A_0010_BK1150_0000_0016_9A12D48F EXTENDS BK1150_A2FCADE7 :
STRUCT
	{attribute addProperty Name "Term_383_KL1002"}
	Term_383_KL1002 : KL1002_BB38DA8F;
END_STRUCT
END_TYPE

// ---- DUTs/IO/Topology/A_0011_BK1150_0000_0017_3F9D1926.TcDUT
{attribute 'GeneratedUsingTerminal: BK1150-0000-0017'}
{attribute addProperty BoxType "BK1150-0000-0017"}
{attribute addProperty Id "Term_384_KL1002KL1002_BB38DA8F0"}
{attribute addProperty CRC "1067260198"}
{attribute addProperty Size "0"}
{attribute addProperty Name "A_0011(BK1150-0000-0017)"}
TYPE A_0011_BK1150_0000_0017_3F9D1926 EXTENDS BK1150_A2FCADE7 :
STRUCT
	{attribute addProperty Name "Term_384_KL1002"}
	Term_384_KL1002 : KL1002_BB38DA8F;
END_STRUCT
END_TYPE

// ---- DUTs/IO/Topology/A_0012_BK1150_0000_0018_69328494.TcDUT
{attribute 'GeneratedUsingTerminal: BK1150-0000-0018'}
{attribute addProperty BoxType "BK1150-0000-0018"}
{attribute addProperty Id "Term_385_KL1002KL1002_BB38DA8F0"}
{attribute addProperty CRC "1764918420"}
{attribute addProperty Size "0"}
{attribute addProperty Name "A_0012(BK1150-0000-0018)"}
TYPE A_0012_BK1150_0000_0018_69328494 EXTENDS BK1150_A2FCADE7 :
STRUCT
	{attribute addProperty Name "Term_385_KL1002"}
	Term_385_KL1002 : KL1002_BB38DA8F;
END_STRUCT
END_TYPE

// ---- DUTs/IO/Topology/A_0013_BK1150_0000_0019_92C22242.TcDUT
{attribute 'GeneratedUsingTerminal: BK1150-0000-0019'}
{attribute addProperty BoxType "BK1150-0000-0019"}
{attribute addProperty Id "Term_386_KL1002KL1002_BB38DA8F0"}
{attribute addProperty CRC "2462196290"}
{attribute addProperty Size "0"}
{attribute addProperty Name "A_0013(BK1150-0000-0019)"}
TYPE A_0013_BK1150_0000_0019_92C22242 EXTENDS BK1150_A2FCADE7 :
STRUCT
	{attribute addProperty Name "Term_386_KL1002"}
	Term_386_KL1002 : KL1002_BB38DA8F;
END_STRUCT
END_TYPE

// ---- DUTs/IO/Topology/A_0016_BK1250_0000_0017_C46DBFF0.TcDUT
{attribute 'GeneratedUsingTerminal: BK1250-0000-0017'}
{attribute addProperty BoxType "BK1250-0000-0017"}
{attribute addProperty Id "Term_387_KL1002KL1002_BB38DA8F0"}
{attribute addProperty CRC "3295526896"}
{attribute addProperty Size "0"}
{attribute addProperty Name "A_0016(BK1250-0000-0017)"}
TYPE A_0016_BK1250_0000_0017_C46DBFF0 EXTENDS BK1250_A2FCADE7 :
STRUCT
	{attribute addProperty Name "Term_387_KL1002"}
	Term_387_KL1002 : KL1002_BB38DA8F;
END_STRUCT
END_TYPE

// ---- DUTs/IO/Topology/Term_19_EK1100_718FBBA4.TcDUT
{attribute 'GeneratedUsingTerminal: EK1100-0000-0018'}
{attribute addProperty BoxType "EK1100-0000-0018"}
{attribute addProperty Id "A_0016_BK1250_0000_0017A_0016_BK1250_0000_0017_C46DBFF00"}
{attribute addProperty CRC "1905245092"}
{attribute addProperty Size "0"}
{attribute addProperty Name "Term 19 (EK1100)"}
TYPE Term_19_EK1100_718FBBA4 EXTENDS EK1100_1FC0878B :
STRUCT
	{attribute addProperty Name "A_0016(BK1250-0000-0017)"}
	{attribute addProperty PreviousPort "Term 19 (EK1100) : B"}
	A_0016_BK1250_0000_0017 : A_0016_BK1250_0000_0017_C46DBFF0;
END_STRUCT
END_TYPE

// ---- DUTs/IO/Topology/A_0018_BK1250_0000_0019_DD1CA4A7.TcDUT
{attribute 'GeneratedUsingTerminal: BK1250-0000-0019'}
{attribute addProperty BoxType "BK1250-0000-0019"}
{attribute addProperty Id "Term_388_KL1002KL1002_BB38DA8F0"}
{attribute addProperty CRC "3709641895"}
{attribute addProperty Size "0"}
{attribute addProperty Name "A_0018(BK1250-0000-0019)"}
TYPE A_0018_BK1250_0000_0019_DD1CA4A7 EXTENDS BK1250_A2FCADE7 :
STRUCT
	{attribute addProperty Name "Term_388_KL1002"}
	Term_388_KL1002 : KL1002_BB38DA8F;
END_STRUCT
END_TYPE

// ---- DUTs/IO/Topology/Term_23_EK1100_08A82DAA.TcDUT
{attribute 'GeneratedUsingTerminal: EK1100-0000-0018'}
{attribute addProperty BoxType "EK1100-0000-0018"}
{attribute addProperty Id "A_0018_BK1250_0000_0019A_0018_BK1250_0000_0019_DD1CA4A70"}
{attribute addProperty CRC "145239466"}
{attribute addProperty Size "0"}
{attribute addProperty Name "Term 23 (EK1100)"}
TYPE Term_23_EK1100_08A82DAA EXTENDS EK1100_1FC0878B :
STRUCT
	{attribute addProperty Name "A_0018(BK1250-0000-0019)"}
	{attribute addProperty PreviousPort "Term 23 (EK1100) : B"}
	A_0018_BK1250_0000_0019 : A_0018_BK1250_0000_0019_DD1CA4A7;
END_STRUCT
END_TYPE

// ---- DUTs/IO/Topology/A_0017_BK1250_0000_0018_8BB33915.TcDUT
{attribute 'GeneratedUsingTerminal: BK1250-0000-0018'}
{attribute addProperty BoxType "BK1250-0000-0018"}
{attribute addProperty Id "Term_389_KL1002KL1002_BB38DA8F0"}
{attribute addProperty CRC "2343778581"}
{attribute addProperty Size "0"}
{attribute addProperty Name "A_0017(BK1250-0000-0018)"}
TYPE A_0017_BK1250_0000_0018_8BB33915 EXTENDS BK1250_A2FCADE7 :
STRUCT
	{attribute addProperty Name "Term_389_KL1002"}
	Term_389_KL1002 : KL1002_BB38DA8F;
END_STRUCT
END_TYPE

// ---- DUTs/IO/Topology/Term_21_EK1100_FD75FF18.TcDUT
{attribute 'GeneratedUsingTerminal: EK1100-0000-0018'}
{attribute addProperty BoxType "EK1100-0000-0018"}
{attribute addProperty Id "A_0017_BK1250_0000_0018A_0017_BK1250_0000_0018_8BB339150"}
{attribute addProperty CRC "4252368664"}
{attribute addProperty Size "0"}
{attribute addProperty Name "Term 21 (EK1100)"}
TYPE Term_21_EK1100_FD75FF18 EXTENDS EK1100_1FC0878B :
STRUCT
	{attribute addProperty Name "A_0017(BK1250-0000-0018)"}
	{attribute addProperty PreviousPort "Term 21 (EK1100) : B"}
	A_0017_BK1250_0000_0018 : A_0017_BK1250_0000_0018_8BB33915;
END_STRUCT
END_TYPE

// ---- DUTs/IO/Topology/A_0019_IL2300_B110_0016_AC908CDE.TcDUT
{attribute 'GeneratedUsingTerminal: IL2300-B110-0016'}
{attribute addProperty BoxType "IL2300-B110-0016"}
{attribute addProperty Id "Term_19KL_D4CFBC220Term_390_Ix1000KL_8EF4D3E90"}
{attribute addProperty CRC "2895154398"}
{attribute addProperty Size "0"}
{attribute addProperty Name "A_0019(IL2300-B110-0016)"}
TYPE A_0019_IL2300_B110_0016_AC908CDE EXTENDS IL2300_A2FCADE7 :
STRUCT
	{attribute addProperty Name "Term_19"}
	Term_19 : KL_D4CFBC22;
	{attribute addProperty Name "Term_390_Ix1000"}
	Term_390_Ix1000 : KL_8EF4D3E9;
END_STRUCT
END_TYPE

// ---- DUTs/IO/Topology/A_0020_IL2300_B110_0017_8C062E24.TcDUT
{attribute 'GeneratedUsingTerminal: IL2300-B110-0017'}
{attribute addProperty BoxType "IL2300-B110-0017"}
{attribute addProperty Id "Term_20KL_D4CFBC220Term_391_Ix1000KL_8EF4D3E90"}
{attribute addProperty CRC "2349215268"}
{attribute addProperty Size "0"}
{attribute addProperty Name "A_0020(IL2300-B110-0017)"}
TYPE A_0020_IL2300_B110_0017_8C062E24 EXTENDS IL2300_A2FCADE7 :
STRUCT
	{attribute addProperty Name "Term_20"}
	Term_20 : KL_D4CFBC22;
	{attribute addProperty Name "Term_391_Ix1000"}
	Term_391_Ix1000 : KL_8EF4D3E9;
END_STRUCT
END_TYPE

// ---- DUTs/IO/Topology/A_0021_IL2301_B110_0016_FF61810D.TcDUT
{attribute 'GeneratedUsingTerminal: IL2301-B110-0016'}
{attribute addProperty BoxType "IL2301-B110-0016"}
{attribute addProperty Id "Term_21KL_D4CFBC220Term_392_Ix1000KL_8EF4D3E90"}
{attribute addProperty CRC "4284580109"}
{attribute addProperty Size "0"}
{attribute addProperty Name "A_0021(IL2301-B110-0016)"}
TYPE A_0021_IL2301_B110_0016_FF61810D EXTENDS IL2301_A2FCADE7 :
STRUCT
	{attribute addProperty Name "Term_21"}
	Term_21 : KL_D4CFBC22;
	{attribute addProperty Name "Term_392_Ix1000"}
	Term_392_Ix1000 : KL_8EF4D3E9;
END_STRUCT
END_TYPE

// ---- DUTs/IO/Topology/A_0022_IL2301_B110_0017_BAC34F2E.TcDUT
{attribute 'GeneratedUsingTerminal: IL2301-B110-0017'}
{attribute addProperty BoxType "IL2301-B110-0017"}
{attribute addProperty Id "Term_22KL_D4CFBC220Term_393_Ix1000KL_8EF4D3E90"}
{attribute addProperty CRC "3133361966"}
{attribute addProperty Size "0"}
{attribute addProperty Name "A_0022(IL2301-B110-0017)"}
TYPE A_0022_IL2301_B110_0017_BAC34F2E EXTENDS IL2301_A2FCADE7 :
STRUCT
	{attribute addProperty Name "Term_22"}
	Term_22 : KL_D4CFBC22;
	{attribute addProperty Name "Term_393_Ix1000"}
	Term_393_Ix1000 : KL_8EF4D3E9;
END_STRUCT
END_TYPE

// ---- DUTs/IO/Topology/A_0023_IL2302_B110_0016_19AEDF5F.TcDUT
{attribute 'GeneratedUsingTerminal: IL2302-B110-0016'}
{attribute addProperty BoxType "IL2302-B110-0016"}
{attribute addProperty Id "Term_23KL_D4CFBC220Term_394_Ix1000KL_8EF4D3E90"}
{attribute addProperty CRC "430890847"}
{attribute addProperty Size "0"}
{attribute addProperty Name "A_0023(IL2302-B110-0016)"}
TYPE A_0023_IL2302_B110_0016_19AEDF5F EXTENDS IL2302_A2FCADE7 :
STRUCT
	{attribute addProperty Name "Term_23"}
	Term_23 : KL_D4CFBC22;
	{attribute addProperty Name "Term_394_Ix1000"}
	Term_394_Ix1000 : KL_8EF4D3E9;
END_STRUCT
END_TYPE

// ---- DUTs/IO/Topology/A_0024_IL2302_B110_0017_E18CEC30.TcDUT
{attribute 'GeneratedUsingTerminal: IL2302-B110-0017'}
{attribute addProperty BoxType "IL2302-B110-0017"}
{attribute addProperty Id "Term_24KL_D4CFBC220Term_395_Ix1000KL_8EF4D3E90"}
{attribute addProperty CRC "3784109104"}
{attribute addProperty Size "0"}
{attribute addProperty Name "A_0024(IL2302-B110-0017)"}
TYPE A_0024_IL2302_B110_0017_E18CEC30 EXTENDS IL2302_A2FCADE7 :
STRUCT
	{attribute addProperty Name "Term_24"}
	Term_24 : KL_D4CFBC22;
	{attribute addProperty Name "Term_395_Ix1000"}
	Term_395_Ix1000 : KL_8EF4D3E9;
END_STRUCT
END_TYPE

// ---- DUTs/IO/Topology/Beckhoff_BKxxxxEK1122_C32C6A5C.TcDUT
{attribute 'GeneratedUsingTerminal: EK1122-0000-0018'}
{attribute addProperty BoxType "EK1122-0000-0018"}
{attribute addProperty Id "Beckhoff_BKxxxxsub_EK1100Beckhoff_BKxxxxsub_EK1100_59A469240A_0001_BK1120_0000_0000A_0001_BK1120_0000_0000_205E65590A_0002_BK1120_0000_0001A_0002_BK1120_0000_0001_76F1F8EB0A_0003_BK1120_0000_0016A_0003_BK1120_0000_0016_8D015E3D0A_0004_BK1120_0000_0017A_0004_BK1120_0000_0017_DBAEC38F0A_0005_BK1120_0000_0018A_0005_BK1120_0000_0018_C2DFD8D80A_0006_BK1120_0000_0019A_0006_BK1120_0000_0019_9470456A0A_0007_BK1120_0000_0020A_0007_BK1120_0000_0020_61E272590A_0008_BK1120_0000_0021A_0008_BK1120_0000_0021_374DEFEB0A_0009_CPXXXX_BK1150_0016A_0009_CPXXXX_BK1150_0016_CCBD493D0A_0010_BK1150_0000_0016A_0010_BK1150_0000_0016_9A12D48F0A_0011_BK1150_0000_0017A_0011_BK1150_0000_0017_3F9D19260A_0012_BK1150_0000_0018A_0012_BK1150_0000_0018_693284940A_0013_BK1150_0000_0019A_0013_BK1150_0000_0019_92C222420Term_19_EK1100Term_19_EK1100_718FBBA40Term_23_EK1100Term_23_EK1100_08A82DAA0Term_21_EK1100Term_21_EK1100_FD75FF180A_0019_IL2300_B110_0016A_0019_IL2300_B110_0016_AC908CDE0A_0020_IL2300_B110_0017A_0020_IL2300_B110_0017_8C062E240A_0021_IL2301_B110_0016A_0021_IL2301_B110_0016_FF61810D0A_0022_IL2301_B110_0017A_0022_IL2301_B110_0017_BAC34F2E0A_0023_IL2302_B110_0016A_0023_IL2302_B110_0016_19AEDF5F0A_0024_IL2302_B110_0017A_0024_IL2302_B110_0017_E18CEC300"}
{attribute addProperty CRC "3274467932"}
{attribute addProperty Size "0"}
{attribute addProperty Name "Beckhoff BKxxxxEK1122"}
TYPE Beckhoff_BKxxxxEK1122_C32C6A5C EXTENDS EK1122_1FC0878B :
STRUCT
	{attribute addProperty Name "Beckhoff BKxxxxsub EK1100"}
	{attribute addProperty PreviousPort "Beckhoff BKxxxxEK1122 : D"}
	Beckhoff_BKxxxxsub_EK1100 : Beckhoff_BKxxxxsub_EK1100_59A46924;
	{attribute addProperty Name "A_0001(BK1120-0000-0000)"}
	{attribute addProperty PreviousPort "Beckhoff BKxxxxEK1122 : B"}
	A_0001_BK1120_0000_0000 : A_0001_BK1120_0000_0000_205E6559;
	{attribute addProperty Name "A_0002(BK1120-0000-0001)"}
	{attribute addProperty PreviousPort "A_0001(BK1120-0000-0000) : B"}
	A_0002_BK1120_0000_0001 : A_0002_BK1120_0000_0001_76F1F8EB;
	{attribute addProperty Name "A_0003(BK1120-0000-0016)"}
	{attribute addProperty PreviousPort "A_0002(BK1120-0000-0001) : B"}
	A_0003_BK1120_0000_0016 : A_0003_BK1120_0000_0016_8D015E3D;
	{attribute addProperty Name "A_0004(BK1120-0000-0017)"}
	{attribute addProperty PreviousPort "A_0003(BK1120-0000-0016) : B"}
	A_0004_BK1120_0000_0017 : A_0004_BK1120_0000_0017_DBAEC38F;
	{attribute addProperty Name "A_0005(BK1120-0000-0018)"}
	{attribute addProperty PreviousPort "A_0004(BK1120-0000-0017) : B"}
	A_0005_BK1120_0000_0018 : A_0005_BK1120_0000_0018_C2DFD8D8;
	{attribute addProperty Name "A_0006(BK1120-0000-0019)"}
	{attribute addProperty PreviousPort "A_0005(BK1120-0000-0018) : B"}
	A_0006_BK1120_0000_0019 : A_0006_BK1120_0000_0019_9470456A;
	{attribute addProperty Name "A_0007(BK1120-0000-0020)"}
	{attribute addProperty PreviousPort "A_0006(BK1120-0000-0019) : B"}
	A_0007_BK1120_0000_0020 : A_0007_BK1120_0000_0020_61E27259;
	{attribute addProperty Name "A_0008(BK1120-0000-0021)"}
	{attribute addProperty PreviousPort "A_0007(BK1120-0000-0020) : B"}
	A_0008_BK1120_0000_0021 : A_0008_BK1120_0000_0021_374DEFEB;
	{attribute addProperty Name "A_0009(CPXXXX-BK1150-0016)"}
	{attribute addProperty PreviousPort "A_0008(BK1120-0000-0021) : B"}
	A_0009_CPXXXX_BK1150_0016 : A_0009_CPXXXX_BK1150_0016_CCBD493D;
	{attribute addProperty Name "A_0010(BK1150-0000-0016)"}
	{attribute addProperty PreviousPort "A_0009(CPXXXX-BK1150-0016) : B"}
	A_0010_BK1150_0000_0016 : A_0010_BK1150_0000_0016_9A12D48F;
	{attribute addProperty Name "A_0011(BK1150-0000-0017)"}
	{attribute addProperty PreviousPort "A_0010(BK1150-0000-0016) : B"}
	A_0011_BK1150_0000_0017 : A_0011_BK1150_0000_0017_3F9D1926;
	{attribute addProperty Name "A_0012(BK1150-0000-0018)"}
	{attribute addProperty PreviousPort "A_0011(BK1150-0000-0017) : B"}
	A_0012_BK1150_0000_0018 : A_0012_BK1150_0000_0018_69328494;
	{attribute addProperty Name "A_0013(BK1150-0000-0019)"}
	{attribute addProperty PreviousPort "A_0012(BK1150-0000-0018) : B"}
	A_0013_BK1150_0000_0019 : A_0013_BK1150_0000_0019_92C22242;
	{attribute addProperty Name "Term 19 (EK1100)"}
	{attribute addProperty PreviousPort "A_0013(BK1150-0000-0019) : B"}
	Term_19_EK1100 : Term_19_EK1100_718FBBA4;
	{attribute addProperty Name "Term 23 (EK1100)"}
	{attribute addProperty PreviousPort "Term 19 (EK1100) : C"}
	Term_23_EK1100 : Term_23_EK1100_08A82DAA;
	{attribute addProperty Name "Term 21 (EK1100)"}
	{attribute addProperty PreviousPort "Term 23 (EK1100) : C"}
	Term_21_EK1100 : Term_21_EK1100_FD75FF18;
	{attribute addProperty Name "A_0019(IL2300-B110-0016)"}
	{attribute addProperty PreviousPort "Term 21 (EK1100) : C"}
	A_0019_IL2300_B110_0016 : A_0019_IL2300_B110_0016_AC908CDE;
	{attribute addProperty Name "A_0020(IL2300-B110-0017)"}
	{attribute addProperty PreviousPort "A_0019(IL2300-B110-0016) : B"}
	A_0020_IL2300_B110_0017 : A_0020_IL2300_B110_0017_8C062E24;
	{attribute addProperty Name "A_0021(IL2301-B110-0016)"}
	{attribute addProperty PreviousPort "A_0020(IL2300-B110-0017) : B"}
	A_0021_IL2301_B110_0016 : A_0021_IL2301_B110_0016_FF61810D;
	{attribute addProperty Name "A_0022(IL2301-B110-0017)"}
	{attribute addProperty PreviousPort "A_0021(IL2301-B110-0016) : B"}
	A_0022_IL2301_B110_0017 : A_0022_IL2301_B110_0017_BAC34F2E;
	{attribute addProperty Name "A_0023(IL2302-B110-0016)"}
	{attribute addProperty PreviousPort "A_0022(IL2301-B110-0017) : B"}
	A_0023_IL2302_B110_0016 : A_0023_IL2302_B110_0016_19AEDF5F;
	{attribute addProperty Name "A_0024(IL2302-B110-0017)"}
	{attribute addProperty PreviousPort "A_0023(IL2302-B110-0016) : B"}
	A_0024_IL2302_B110_0017 : A_0024_IL2302_B110_0017_E18CEC30;
END_STRUCT
END_TYPE

// ---- DUTs/IO/Topology/A_0015_BK1250_0000_0016_5F4E76F7.TcDUT
{attribute 'GeneratedUsingTerminal: BK1250-0000-0016'}
{attribute addProperty BoxType "BK1250-0000-0016"}
{attribute addProperty Id "Term_396_KL1002KL1002_BB38DA8F0"}
{attribute addProperty CRC "1598977783"}
{attribute addProperty Size "0"}
{attribute addProperty Name "A_0015(BK1250-0000-0016)"}
TYPE A_0015_BK1250_0000_0016_5F4E76F7 EXTENDS BK1250_A2FCADE7 :
STRUCT
	{attribute addProperty Name "Term_396_KL1002"}
	Term_396_KL1002 : KL1002_BB38DA8F;
END_STRUCT
END_TYPE

// ---- DUTs/IO/Topology/Beckhoff_BKxxxx_735133AB.TcDUT
{attribute 'GeneratedUsingTerminal: EK1100-0000-0018'}
{attribute addProperty BoxType "EK1100-0000-0018"}
{attribute addProperty Id "Beckhoff_BKxxxxEK1122Beckhoff_BKxxxxEK1122_C32C6A5C0A_0015_BK1250_0000_0016A_0015_BK1250_0000_0016_5F4E76F70"}
{attribute addProperty CRC "1934701483"}
{attribute addProperty Size "0"}
{attribute addProperty Name "Beckhoff BKxxxx"}
TYPE Beckhoff_BKxxxx_735133AB EXTENDS EK1100_1FC0878B :
STRUCT
	{attribute addProperty Name "Beckhoff BKxxxxEK1122"}
	{attribute addProperty PreviousPort "Beckhoff BKxxxx : B"}
	Beckhoff_BKxxxxEK1122 : Beckhoff_BKxxxxEK1122_C32C6A5C;
	{attribute addProperty Name "A_0015(BK1250-0000-0016)"}
	{attribute addProperty PreviousPort "Beckhoff BKxxxxEK1122 : C"}
	A_0015_BK1250_0000_0016 : A_0015_BK1250_0000_0016_5F4E76F7;
END_STRUCT
END_TYPE

// ---- DUTs/IO/Topology/A_0006_CU1128_0000_0002_093CCA2E.TcDUT
{attribute 'GeneratedUsingTerminal: CU1128-0000-0002'}
{attribute addProperty BoxType "CU1128-0000-0002"}
{attribute addProperty Id "A_0007_CU1521_0010_0000CU1521_1FC0878B2A_0008_CU1561_0000_0000CU1561_1FC0878B2A_0009_CU2508_0000_0000CU2508_1FC0878B2A_0010_CU2508_0000_0016CU2508_EEB2FEF410A_0011_CU2508_0000_0017CU2508_6BF2ACBC32A_0012_CU2508_0000_0018CU2508_6BF2ACBC32A_0013_CU2508_0000_0019CU2508_6BF2ACBC32A_0006_CU1128_0000_0002_2_CU1128_BCU1128_1FC0878B2A_0006_CU1128_0000_0002_3_CU1128_CCU1128_1FC0878B2"}
{attribute addProperty CRC "154978862"}
{attribute addProperty Size "116"}
{attribute addProperty Name "A_0006(CU1128-0000-0002)"}
TYPE A_0006_CU1128_0000_0002_093CCA2E EXTENDS CU1128_1FC0878B :
STRUCT
	{attribute addProperty Name "A_0007(CU1521-0010-0000)"}
	{attribute addProperty PreviousPort "A_0006(CU1128-0000-0002) : D"}
	A_0007_CU1521_0010_0000 : CU1521_1FC0878B;
	{attribute addProperty Name "A_0008(CU1561-0000-0000)"}
	{attribute addProperty PreviousPort "A_0007(CU1521-0010-0000) : B"}
	A_0008_CU1561_0000_0000 : CU1561_1FC0878B;
	{attribute addProperty Name "A_0009(CU2508-0000-0000)"}
	{attribute addProperty PreviousPort "A_0008(CU1561-0000-0000) : B"}
	A_0009_CU2508_0000_0000 : CU2508_1FC0878B;
	{attribute addProperty Name "A_0010(CU2508-0000-0016)"}
	{attribute addProperty PreviousPort "A_0009(CU2508-0000-0000) : B"}
	A_0010_CU2508_0000_0016 : CU2508_EEB2FEF4;
	{attribute addProperty Name "A_0011(CU2508-0000-0017)"}
	{attribute addProperty PreviousPort "A_0010(CU2508-0000-0016) : B"}
	A_0011_CU2508_0000_0017 : CU2508_6BF2ACBC;
	{attribute addProperty Name "A_0012(CU2508-0000-0018)"}
	{attribute addProperty PreviousPort "A_0011(CU2508-0000-0017) : B"}
	A_0012_CU2508_0000_0018 : CU2508_6BF2ACBC;
	{attribute addProperty Name "A_0013(CU2508-0000-0019)"}
	{attribute addProperty PreviousPort "A_0012(CU2508-0000-0018) : B"}
	A_0013_CU2508_0000_0019 : CU2508_6BF2ACBC;
	{attribute addProperty Name "A_0006(CU1128-0000-0002)_2 (CU1128-B)"}
	{attribute addProperty PreviousPort "A_0006(CU1128-0000-0002) : C"}
	A_0006_CU1128_0000_0002_2_CU1128_B : CU1128_1FC0878B;
	{attribute addProperty Name "A_0006(CU1128-0000-0002)_3 (CU1128-C)"}
	{attribute addProperty PreviousPort "A_0006(CU1128-0000-0002)_2 (CU1128-B) : C"}
	A_0006_CU1128_0000_0002_3_CU1128_C : CU1128_1FC0878B;
END_STRUCT
END_TYPE

// ---- DUTs/IO/Topology/A_0005_CU1128_0000_0001_8DEFD527.TcDUT
{attribute 'GeneratedUsingTerminal: CU1128-0000-0001'}
{attribute addProperty BoxType "CU1128-0000-0001"}
{attribute addProperty Id "A_0006_CU1128_0000_0002A_0006_CU1128_0000_0002_093CCA2E116A_0005_CU1128_0000_0001_2_CU1128_BCU1128_1FC0878B2A_0005_CU1128_0000_0001_3_CU1128_CCU1128_1FC0878B2"}
{attribute addProperty CRC "2381305127"}
{attribute addProperty Size "120"}
{attribute addProperty Name "A_0005(CU1128-0000-0001)"}
TYPE A_0005_CU1128_0000_0001_8DEFD527 EXTENDS CU1128_1FC0878B :
STRUCT
	{attribute addProperty Name "A_0006(CU1128-0000-0002)"}
	{attribute addProperty PreviousPort "A_0005(CU1128-0000-0001) : D"}
	A_0006_CU1128_0000_0002 : A_0006_CU1128_0000_0002_093CCA2E;
	{attribute addProperty Name "A_0005(CU1128-0000-0001)_2 (CU1128-B)"}
	{attribute addProperty PreviousPort "A_0005(CU1128-0000-0001) : C"}
	A_0005_CU1128_0000_0001_2_CU1128_B : CU1128_1FC0878B;
	{attribute addProperty Name "A_0005(CU1128-0000-0001)_3 (CU1128-C)"}
	{attribute addProperty PreviousPort "A_0005(CU1128-0000-0001)_2 (CU1128-B) : C"}
	A_0005_CU1128_0000_0001_3_CU1128_C : CU1128_1FC0878B;
END_STRUCT
END_TYPE

// ---- DUTs/IO/Topology/A_0004_CU1128_0000_0000_2F60DA9F.TcDUT
{attribute 'GeneratedUsingTerminal: CU1128--0000'}
{attribute addProperty BoxType "CU1128--0000"}
{attribute addProperty Id "A_0005_CU1128_0000_0001A_0005_CU1128_0000_0001_8DEFD527120A_0004_CU1128_0000_0000_2_CU1128_BCU1128_1FC0878B2A_0004_CU1128_0000_0000_3_CU1128_CCU1128_1FC0878B2"}
{attribute addProperty CRC "794876575"}
{attribute addProperty Size "124"}
{attribute addProperty Name "A_0004(CU1128-0000-0000)"}
TYPE A_0004_CU1128_0000_0000_2F60DA9F EXTENDS CU1128_1FC0878B :
STRUCT
	{attribute addProperty Name "A_0005(CU1128-0000-0001)"}
	{attribute addProperty PreviousPort "A_0004(CU1128-0000-0000) : D"}
	A_0005_CU1128_0000_0001 : A_0005_CU1128_0000_0001_8DEFD527;
	{attribute addProperty Name "A_0004(CU1128-0000-0000)_2 (CU1128-B)"}
	{attribute addProperty PreviousPort "A_0004(CU1128-0000-0000) : C"}
	A_0004_CU1128_0000_0000_2_CU1128_B : CU1128_1FC0878B;
	{attribute addProperty Name "A_0004(CU1128-0000-0000)_3 (CU1128-C)"}
	{attribute addProperty PreviousPort "A_0004(CU1128-0000-0000)_2 (CU1128-B) : C"}
	A_0004_CU1128_0000_0000_3_CU1128_C : CU1128_1FC0878B;
END_STRUCT
END_TYPE

// ---- DUTs/IO/Topology/A_0003_CU1124_0000_0016_CE6B0448.TcDUT
{attribute 'GeneratedUsingTerminal: CU1124-0000-0016'}
{attribute addProperty BoxType "CU1124-0000-0016"}
{attribute addProperty Id "A_0004_CU1128_0000_0000A_0004_CU1128_0000_0000_2F60DA9F124"}
{attribute addProperty CRC "3463119944"}
{attribute addProperty Size "124"}
{attribute addProperty Name "A_0003(CU1124-0000-0016)"}
TYPE A_0003_CU1124_0000_0016_CE6B0448 EXTENDS CU1124_1FC0878B :
STRUCT
	{attribute addProperty Name "A_0004(CU1128-0000-0000)"}
	{attribute addProperty PreviousPort "A_0003(CU1124-0000-0016) : D"}
	A_0004_CU1128_0000_0000 : A_0004_CU1128_0000_0000_2F60DA9F;
END_STRUCT
END_TYPE

// ---- DUTs/IO/Topology/A_0002_CU1123_0010_0016_E68B3D99.TcDUT
{attribute 'GeneratedUsingTerminal: CU1123-0010-0016'}
{attribute addProperty BoxType "CU1123-0010-0016"}
{attribute addProperty Id "A_0003_CU1124_0000_0016A_0003_CU1124_0000_0016_CE6B0448124"}
{attribute addProperty CRC "3867884953"}
{attribute addProperty Size "124"}
{attribute addProperty Name "A_0002(CU1123-0010-0016)"}
TYPE A_0002_CU1123_0010_0016_E68B3D99 EXTENDS CU1123_1FC0878B :
STRUCT
	{attribute addProperty Name "A_0003(CU1124-0000-0016)"}
	{attribute addProperty PreviousPort "A_0002(CU1123-0010-0016) : D"}
	A_0003_CU1124_0000_0016 : A_0003_CU1124_0000_0016_CE6B0448;
END_STRUCT
END_TYPE

// ---- DUTs/IO/Topology/A_0001_CU1123_0000_0016_30E128CC.TcDUT
{attribute 'GeneratedUsingTerminal: CU1123-0000-0016'}
{attribute addProperty BoxType "CU1123-0000-0016"}
{attribute addProperty Id "A_0002_CU1123_0010_0016A_0002_CU1123_0010_0016_E68B3D99124"}
{attribute addProperty CRC "820062412"}
{attribute addProperty Size "124"}
{attribute addProperty Name "A_0001(CU1123-0000-0016)"}
TYPE A_0001_CU1123_0000_0016_30E128CC EXTENDS CU1123_1FC0878B :
STRUCT
	{attribute addProperty Name "A_0002(CU1123-0010-0016)"}
	{attribute addProperty PreviousPort "A_0001(CU1123-0000-0016) : D"}
	A_0002_CU1123_0010_0016 : A_0002_CU1123_0010_0016_E68B3D99;
END_STRUCT
END_TYPE

// ---- DUTs/IO/Topology/Beckhoff_CUxxxxEK1122_BE344318.TcDUT
{attribute 'GeneratedUsingTerminal: EK1122-0000-0018'}
{attribute addProperty BoxType "EK1122-0000-0018"}
{attribute addProperty Id "Beckhoff_CUxxxxsub_EK1100EK1100_1FC0878B2A_0001_CU1123_0000_0016A_0001_CU1123_0000_0016_30E128CC124"}
{attribute addProperty CRC "3191096088"}
{attribute addProperty Size "126"}
{attribute addProperty Name "Beckhoff CUxxxxEK1122"}
TYPE Beckhoff_CUxxxxEK1122_BE344318 EXTENDS EK1122_1FC0878B :
STRUCT
	{attribute addProperty Name "Beckhoff CUxxxxsub EK1100"}
	{attribute addProperty PreviousPort "Beckhoff CUxxxxEK1122 : D"}
	Beckhoff_CUxxxxsub_EK1100 : EK1100_1FC0878B;
	{attribute addProperty Name "A_0001(CU1123-0000-0016)"}
	{attribute addProperty PreviousPort "Beckhoff CUxxxxsub EK1100 : C"}
	A_0001_CU1123_0000_0016 : A_0001_CU1123_0000_0016_30E128CC;
END_STRUCT
END_TYPE

// ---- DUTs/IO/Topology/Beckhoff_CUxxxx_E9AD9532.TcDUT
{attribute 'GeneratedUsingTerminal: EK1100-0000-0018'}
{attribute addProperty BoxType "EK1100-0000-0018"}
{attribute addProperty Id "Beckhoff_CUxxxxEK1122Beckhoff_CUxxxxEK1122_BE344318126"}
{attribute addProperty CRC "3920467250"}
{attribute addProperty Size "126"}
{attribute addProperty Name "Beckhoff CUxxxx"}
TYPE Beckhoff_CUxxxx_E9AD9532 EXTENDS EK1100_1FC0878B :
STRUCT
	{attribute addProperty Name "Beckhoff CUxxxxEK1122"}
	{attribute addProperty PreviousPort "Beckhoff CUxxxx : B"}
	Beckhoff_CUxxxxEK1122 : Beckhoff_CUxxxxEK1122_BE344318;
END_STRUCT
END_TYPE

// ---- DUTs/IO/Topology/Beckhoff_CXxxxxEK1122_ADC91C0D.TcDUT
{attribute 'GeneratedUsingTerminal: EK1122-0000-0018'}
{attribute addProperty BoxType "EK1122-0000-0018"}
{attribute addProperty Id "Beckhoff_CXxxxxsub_EK1100EK1100_1FC0878B2A_0001_CX1100_0004_0000CX1100_1FC0878B2A_0003_CX1100_0004_0002CX1100_1FC0878B2A_0004_CX5010_EtherCAT_slaveCX5010_EtherCAT_slave_FEF7A27A20A_0005_CX5010_EtherCAT_slaveCX5010_EtherCAT_slave_FEF7A27A20A_0006_CX5020_EtherCAT_slaveCX5020_EtherCAT_slave_FEF7A27A20A_0007_CX5020_EtherCAT_slaveCX5020_EtherCAT_slave_FEF7A27A20A_0008_CX8010_EtherCAT_slaveCX8010_EtherCAT_slave_FEF7A27A20A_0009_CX8010_EtherCAT_slaveCX8010_EtherCAT_slave_FEF7A27A20A_0010_CX8110_EtherCAT_slaveCX8110_EtherCAT_slave_FEF7A27A20A_0011_CX2020_EtherCAT_slaveCX2020_EtherCAT_slave_FEF7A27A20A_0012_CX2020_EtherCAT_slaveCX2020_EtherCAT_slave_FEF7A27A20A_0013_CX2020_EtherCAT_slaveCX2020_EtherCAT_slave_FEF7A27A20A_0014_CX2030_EtherCAT_slaveCX2030_EtherCAT_slave_FEF7A27A20A_0015_CX2030_EtherCAT_slaveCX2030_EtherCAT_slave_FEF7A27A20A_0016_CX2030_EtherCAT_slaveCX2030_EtherCAT_slave_FEF7A27A20A_0017_CX2033_EtherCAT_slaveCX2033_EtherCAT_slave_FEF7A27A20A_0018_CX2040_EtherCAT_slaveCX2040_EtherCAT_slave_FEF7A27A20A_0019_CX2040_EtherCAT_slaveCX2040_EtherCAT_slave_FEF7A27A20A_0020_CX2040_EtherCAT_slaveCX2040_EtherCAT_slave_FEF7A27A20A_0021_CX2042_EtherCAT_slaveCX2042_EtherCAT_slave_FEF7A27A20A_0022_CX2043_EtherCAT_slaveCX2043_EtherCAT_slave_FEF7A27A20A_0023_CX2062_EtherCAT_slaveCX2062_EtherCAT_slave_FEF7A27A20A_0024_CX2072_EtherCAT_slaveCX2072_EtherCAT_slave_FEF7A27A20A_0025_CX9020_EtherCAT_slaveCX9020_EtherCAT_slave_FEF7A27A20A_0026_CX9020_EtherCAT_slaveCX9020_EtherCAT_slave_FEF7A27A20A_0027_CX5120_EtherCAT_slaveCX5120_EtherCAT_slave_FEF7A27A20A_0028_CX5130_EtherCAT_slaveCX5130_EtherCAT_slave_FEF7A27A20A_0029_CX5140_EtherCAT_slaveCX5140_EtherCAT_slave_FEF7A27A20A_0030_CX5230_EtherCAT_slaveCX5230_EtherCAT_slave_FEF7A27A20A_0031_CX5240_EtherCAT_slaveCX5240_EtherCAT_slave_FEF7A27A20A_0002_CX1100_0004_0001CX1100_1FC0878B2"}
{attribute addProperty CRC "2915638285"}
{attribute addProperty Size "568"}
{attribute addProperty Name "Beckhoff CXxxxxEK1122"}
TYPE Beckhoff_CXxxxxEK1122_ADC91C0D EXTENDS EK1122_1FC0878B :
STRUCT
	{attribute addProperty Name "Beckhoff CXxxxxsub EK1100"}
	{attribute addProperty PreviousPort "Beckhoff CXxxxxEK1122 : D"}
	Beckhoff_CXxxxxsub_EK1100 : EK1100_1FC0878B;
	{attribute addProperty Name "A_0001(CX1100-0004-0000)"}
	{attribute addProperty PreviousPort "Beckhoff CXxxxxsub EK1100 : C"}
	A_0001_CX1100_0004_0000 : CX1100_1FC0878B;
	{attribute addProperty Name "A_0003(CX1100-0004-0002)"}
	{attribute addProperty PreviousPort "A_0001(CX1100-0004-0000) : C"}
	A_0003_CX1100_0004_0002 : CX1100_1FC0878B;
	{attribute addProperty Name "A_0004 (CX5010 EtherCAT slave)"}
	{attribute addProperty PreviousPort "Beckhoff CXxxxxEK1122 : B"}
	A_0004_CX5010_EtherCAT_slave : CX5010_EtherCAT_slave_FEF7A27A;
	{attribute addProperty Name "A_0005 (CX5010 EtherCAT slave)"}
	{attribute addProperty PreviousPort "A_0004 (CX5010 EtherCAT slave) : B"}
	A_0005_CX5010_EtherCAT_slave : CX5010_EtherCAT_slave_FEF7A27A;
	{attribute addProperty Name "A_0006 (CX5020 EtherCAT slave)"}
	{attribute addProperty PreviousPort "A_0005 (CX5010 EtherCAT slave) : B"}
	A_0006_CX5020_EtherCAT_slave : CX5020_EtherCAT_slave_FEF7A27A;
	{attribute addProperty Name "A_0007 (CX5020 EtherCAT slave)"}
	{attribute addProperty PreviousPort "A_0006 (CX5020 EtherCAT slave) : B"}
	A_0007_CX5020_EtherCAT_slave : CX5020_EtherCAT_slave_FEF7A27A;
	{attribute addProperty Name "A_0008 (CX8010 EtherCAT slave)"}
	{attribute addProperty PreviousPort "A_0007 (CX5020 EtherCAT slave) : B"}
	A_0008_CX8010_EtherCAT_slave : CX8010_EtherCAT_slave_FEF7A27A;
	{attribute addProperty Name "A_0009 (CX8010 EtherCAT slave)"}
	{attribute addProperty PreviousPort "A_0008 (CX8010 EtherCAT slave) : B"}
	A_0009_CX8010_EtherCAT_slave : CX8010_EtherCAT_slave_FEF7A27A;
	{attribute addProperty Name "A_0010 (CX8110 EtherCAT slave)"}
	{attribute addProperty PreviousPort "A_0009 (CX8010 EtherCAT slave) : B"}
	A_0010_CX8110_EtherCAT_slave : CX8110_EtherCAT_slave_FEF7A27A;
	{attribute addProperty Name "A_0011 (CX2020 EtherCAT slave)"}
	{attribute addProperty PreviousPort "A_0010 (CX8110 EtherCAT slave) : B"}
	A_0011_CX2020_EtherCAT_slave : CX2020_EtherCAT_slave_FEF7A27A;
	{attribute addProperty Name "A_0012 (CX2020 EtherCAT slave)"}
	{attribute addProperty PreviousPort "A_0011 (CX2020 EtherCAT slave) : B"}
	A_0012_CX2020_EtherCAT_slave : CX2020_EtherCAT_slave_FEF7A27A;
	{attribute addProperty Name "A_0013 (CX2020 EtherCAT slave)"}
	{attribute addProperty PreviousPort "A_0012 (CX2020 EtherCAT slave) : B"}
	A_0013_CX2020_EtherCAT_slave : CX2020_EtherCAT_slave_FEF7A27A;
	{attribute addProperty Name "A_0014 (CX2030 EtherCAT slave)"}
	{attribute addProperty PreviousPort "A_0013 (CX2020 EtherCAT slave) : B"}
	A_0014_CX2030_EtherCAT_slave : CX2030_EtherCAT_slave_FEF7A27A;
	{attribute addProperty Name "A_0015 (CX2030 EtherCAT slave)"}
	{attribute addProperty PreviousPort "A_0014 (CX2030 EtherCAT slave) : B"}
	A_0015_CX2030_EtherCAT_slave : CX2030_EtherCAT_slave_FEF7A27A;
	{attribute addProperty Name "A_0016 (CX2030 EtherCAT slave)"}
	{attribute addProperty PreviousPort "A_0015 (CX2030 EtherCAT slave) : B"}
	A_0016_CX2030_EtherCAT_slave : CX2030_EtherCAT_slave_FEF7A27A;
	{attribute addProperty Name "A_0017 (CX2033 EtherCAT slave)"}
	{attribute addProperty PreviousPort "A_0016 (CX2030 EtherCAT slave) : B"}
	A_0017_CX2033_EtherCAT_slave : CX2033_EtherCAT_slave_FEF7A27A;
	{attribute addProperty Name "A_0018 (CX2040 EtherCAT slave)"}
	{attribute addProperty PreviousPort "A_0017 (CX2033 EtherCAT slave) : B"}
	A_0018_CX2040_EtherCAT_slave : CX2040_EtherCAT_slave_FEF7A27A;
	{attribute addProperty Name "A_0019 (CX2040 EtherCAT slave)"}
	{attribute addProperty PreviousPort "A_0018 (CX2040 EtherCAT slave) : B"}
	A_0019_CX2040_EtherCAT_slave : CX2040_EtherCAT_slave_FEF7A27A;
	{attribute addProperty Name "A_0020 (CX2040 EtherCAT slave)"}
	{attribute addProperty PreviousPort "A_0019 (CX2040 EtherCAT slave) : B"}
	A_0020_CX2040_EtherCAT_slave : CX2040_EtherCAT_slave_FEF7A27A;
	{attribute addProperty Name "A_0021 (CX2042 EtherCAT slave)"}
	{attribute addProperty PreviousPort "A_0020 (CX2040 EtherCAT slave) : B"}
	A_0021_CX2042_EtherCAT_slave : CX2042_EtherCAT_slave_FEF7A27A;
	{attribute addProperty Name "A_0022 (CX2043 EtherCAT slave)"}
	{attribute addProperty PreviousPort "A_0021 (CX2042 EtherCAT slave) : B"}
	A_0022_CX2043_EtherCAT_slave : CX2043_EtherCAT_slave_FEF7A27A;
	{attribute addProperty Name "A_0023 (CX2062 EtherCAT slave)"}
	{attribute addProperty PreviousPort "A_0022 (CX2043 EtherCAT slave) : B"}
	A_0023_CX2062_EtherCAT_slave : CX2062_EtherCAT_slave_FEF7A27A;
	{attribute addProperty Name "A_0024 (CX2072 EtherCAT slave)"}
	{attribute addProperty PreviousPort "A_0023 (CX2062 EtherCAT slave) : B"}
	A_0024_CX2072_EtherCAT_slave : CX2072_EtherCAT_slave_FEF7A27A;
	{attribute addProperty Name "A_0025 (CX9020 EtherCAT slave)"}
	{attribute addProperty PreviousPort "A_0024 (CX2072 EtherCAT slave) : B"}
	A_0025_CX9020_EtherCAT_slave : CX9020_EtherCAT_slave_FEF7A27A;
	{attribute addProperty Name "A_0026 (CX9020 EtherCAT slave)"}
	{attribute addProperty PreviousPort "A_0025 (CX9020 EtherCAT slave) : B"}
	A_0026_CX9020_EtherCAT_slave : CX9020_EtherCAT_slave_FEF7A27A;
	{attribute addProperty Name "A_0027 (CX5120 EtherCAT slave)"}
	{attribute addProperty PreviousPort "A_0026 (CX9020 EtherCAT slave) : B"}
	A_0027_CX5120_EtherCAT_slave : CX5120_EtherCAT_slave_FEF7A27A;
	{attribute addProperty Name "A_0028 (CX5130 EtherCAT slave)"}
	{attribute addProperty PreviousPort "A_0027 (CX5120 EtherCAT slave) : B"}
	A_0028_CX5130_EtherCAT_slave : CX5130_EtherCAT_slave_FEF7A27A;
	{attribute addProperty Name "A_0029 (CX5140 EtherCAT slave)"}
	{attribute addProperty PreviousPort "A_0028 (CX5130 EtherCAT slave) : B"}
	A_0029_CX5140_EtherCAT_slave : CX5140_EtherCAT_slave_FEF7A27A;
	{attribute addProperty Name "A_0030 (CX5230 EtherCAT slave)"}
	{attribute addProperty PreviousPort "A_0029 (CX5140 EtherCAT slave) : B"}
	A_0030_CX5230_EtherCAT_slave : CX5230_EtherCAT_slave_FEF7A27A;
	{attribute addProperty Name "A_0031 (CX5240 EtherCAT slave)"}
	{attribute addProperty PreviousPort "A_0030 (CX5230 EtherCAT slave) : B"}
	A_0031_CX5240_EtherCAT_slave : CX5240_EtherCAT_slave_FEF7A27A;
	{attribute addProperty Name "A_0002(CX1100-0004-0001)"}
	{attribute addProperty PreviousPort "A_0031 (CX5240 EtherCAT slave) : B"}
	A_0002_CX1100_0004_0001 : CX1100_1FC0878B;
END_STRUCT
END_TYPE

// ---- DUTs/IO/Topology/Beckhoff_CXxxxx_7C0A3C1E.TcDUT
{attribute 'GeneratedUsingTerminal: EK1100-0000-0018'}
{attribute addProperty BoxType "EK1100-0000-0018"}
{attribute addProperty Id "Beckhoff_CXxxxxEK1122Beckhoff_CXxxxxEK1122_ADC91C0D568"}
{attribute addProperty CRC "2081045534"}
{attribute addProperty Size "568"}
{attribute addProperty Name "Beckhoff CXxxxx"}
TYPE Beckhoff_CXxxxx_7C0A3C1E EXTENDS EK1100_1FC0878B :
STRUCT
	{attribute addProperty Name "Beckhoff CXxxxxEK1122"}
	{attribute addProperty PreviousPort "Beckhoff CXxxxx : B"}
	Beckhoff_CXxxxxEK1122 : Beckhoff_CXxxxxEK1122_ADC91C0D;
END_STRUCT
END_TYPE

